(* CoDeSys 2.3.9.50 project: 10A.pr6 *)
(* Libraries: STANDARD.LB6 5.6.98 12:03:02 *)

(* POU MAIN, LD *)
PROGRAM MAIN
VAR
	reset AT %QX7.7: BOOL
	Light_Sequence: ARRAY [0..7,1..4] OF INT := 1,3,3,3,2,3,2,3,3,3,1,3,3,2,2,3,3,1,3,3,3,2,3,2,3,3,3,1,2,3,3,2;
	Start AT %IX0.0: BOOL;
	Stop AT %IX0.1: BOOL;
	ProcessON AT %QX0.0: BOOL;
	T1: TON;
	C1: CTU;
	East_Green AT %QX2.0: BOOL;
	East_Yellow AT %QX2.1: BOOL;
	East_Red AT %QX2.2: BOOL;
	West_Green AT %QX3.0: BOOL;
	West_Yellow AT %QX3.1: BOOL;
	West_Red AT %QX3.2: BOOL;
	North_Green AT %QX4.0: BOOL;
	North_Yellow AT %QX4.1: BOOL;
	North_Red AT %QX4.2: BOOL;
	South_Green AT %QX5.0: BOOL;
	South_Yellow AT %QX5.1: BOOL;
	South_Red AT %QX5.2: BOOL;
END_VAR
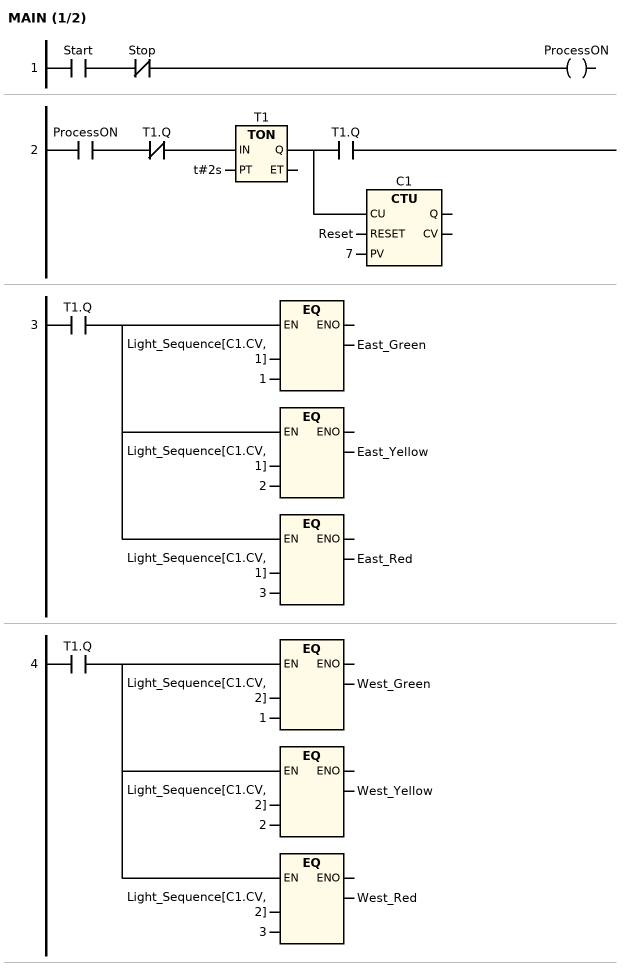
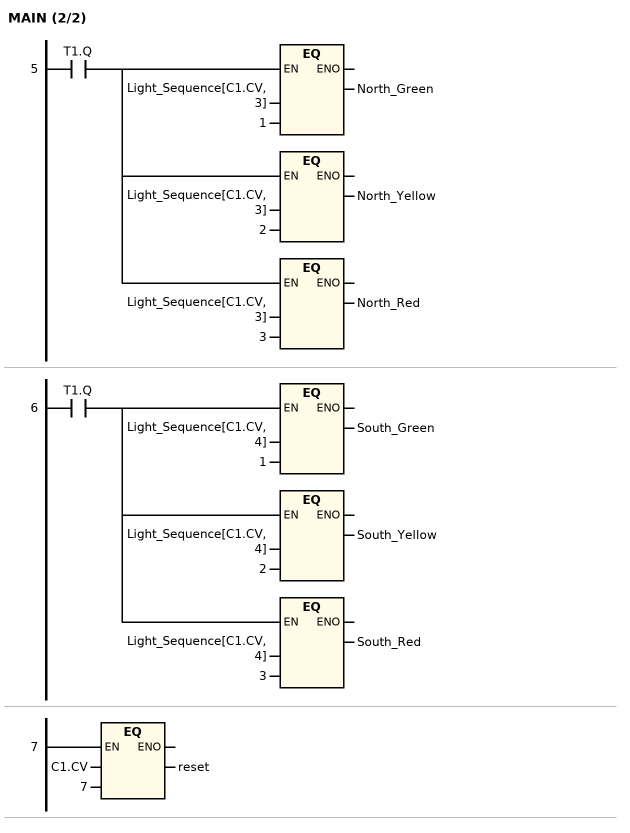
_LD_ (* Ladder Diagram *)
NETWORK 1
	[Start] - [/Stop] --- (ProcessON)
NETWORK 2
	[ProcessON] - [/T1.Q] - T1:TON(IN: *, PT: t#2s) - { [T1.Q] | C1:CTU(CU: *, RESET: Reset, PV: 7) }
NETWORK 3
	[T1.Q]
		EN --- EQ(Light_Sequence[C1.CV,1], 1) => East_Green
		EN --- EQ(Light_Sequence[C1.CV,1], 2) => East_Yellow
		EN --- EQ(Light_Sequence[C1.CV,1], 3) => East_Red
NETWORK 4
	[T1.Q]
		EN --- EQ(Light_Sequence[C1.CV,2], 1) => West_Green
		EN --- EQ(Light_Sequence[C1.CV,2], 2) => West_Yellow
		EN --- EQ(Light_Sequence[C1.CV,2], 3) => West_Red
NETWORK 5
	[T1.Q]
		EN --- EQ(Light_Sequence[C1.CV,3], 1) => North_Green
		EN --- EQ(Light_Sequence[C1.CV,3], 2) => North_Yellow
		EN --- EQ(Light_Sequence[C1.CV,3], 3) => North_Red
NETWORK 6
	[T1.Q]
		EN --- EQ(Light_Sequence[C1.CV,4], 1) => South_Green
		EN --- EQ(Light_Sequence[C1.CV,4], 2) => South_Yellow
		EN --- EQ(Light_Sequence[C1.CV,4], 3) => South_Red
NETWORK 7
	*
		EN --- EQ(C1.CV, 7) => reset
_END_LD_
(* the same logic as Structured Text *)
(* Network 1 *)
ProcessON := Start AND NOT Stop;
(* Network 2 *)
T1(IN := ProcessON AND NOT T1.Q, PT := t#2s);
C1(CU := T1.Q, RESET := Reset, PV := 7);
(* Network 3 *)
IF T1.Q THEN
	East_Green := (Light_Sequence[C1.CV,1]) = 1;
	East_Yellow := (Light_Sequence[C1.CV,1]) = 2;
	East_Red := (Light_Sequence[C1.CV,1]) = 3;
END_IF;
(* Network 4 *)
IF T1.Q THEN
	West_Green := (Light_Sequence[C1.CV,2]) = 1;
	West_Yellow := (Light_Sequence[C1.CV,2]) = 2;
	West_Red := (Light_Sequence[C1.CV,2]) = 3;
END_IF;
(* Network 5 *)
IF T1.Q THEN
	North_Green := (Light_Sequence[C1.CV,3]) = 1;
	North_Yellow := (Light_Sequence[C1.CV,3]) = 2;
	North_Red := (Light_Sequence[C1.CV,3]) = 3;
END_IF;
(* Network 6 *)
IF T1.Q THEN
	South_Green := (Light_Sequence[C1.CV,4]) = 1;
	South_Yellow := (Light_Sequence[C1.CV,4]) = 2;
	South_Red := (Light_Sequence[C1.CV,4]) = 3;
END_IF;
(* Network 7 *)
reset := C1.CV = 7;
END_PROGRAM

(* Visualisation traffic_Light
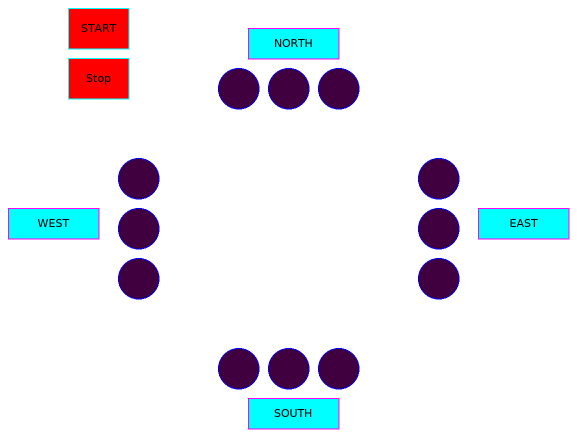
ellipse at (310,80)-(351,121): alarm colour if %qx4.2
ellipse at (310,360)-(351,401): alarm colour if %qx5.0
ellipse at (410,360)-(451,401): alarm colour if %qx5.2
ellipse at (360,360)-(401,401): alarm colour if %qx5.1
ellipse at (510,270)-(551,311): alarm colour if %QX2.0
ellipse at (510,220)-(551,261): alarm colour if %qx2.1
ellipse at (510,170)-(551,211): alarm colour if %qx2.2
ellipse at (210,170)-(251,211): alarm colour if %qx3.0
ellipse at (210,270)-(251,311): alarm colour if %qx3.2
ellipse at (210,220)-(251,261): alarm colour if %qx3.1
ellipse at (410,80)-(451,121): alarm colour if %qx4.0
ellipse at (360,80)-(401,121): alarm colour if %qx4.1
rounded rectangle at (340,40)-(431,71): text "NORTH"
rounded rectangle at (100,220)-(191,251): text "WEST"
rounded rectangle at (340,410)-(431,441): text "SOUTH"
rounded rectangle at (570,220)-(661,251): text "EAST"
rectangle at (160,20)-(221,61): text "START"; alarm colour if %IX0.0; toggles %ix0.0
rectangle at (160,70)-(221,111): text "Stop"; alarm colour if %IX0.1; toggles %IX0.1
*)
